FUNCTION_BLOCK Machine EXTENDS FB_PackML_BaseModule
VAR
END_VAR

METHOD PROTECTED HMIPermissions
AllowHMIControl(ThisModuleOnly := TRUE);
END_METHOD

END_FUNCTION_BLOCK

(* stored: Version 1.1.0.1
   POU Machine: Id {f6ae2cbe-173e-4d75-bb5e-334498954288}, SpecialFunc None
   Method HMIPermissions: Id {01f1aea6-e802-48f8-abd4-50a2a3d31fba} *)
